ABB RobotStudio station: voice_control_abb.rspag

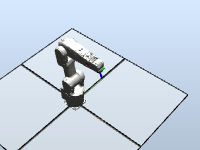
--- station ---
Station Station (saved by RobotStudio 6.7.7850.130)
Controller demo
  mechanical unit ROB_1: IRB1200_5_90_STD_02_2, 6 joints, base frame (0, 0, 0) mm
Layout (positions relative to the parent item):
  - IRB1200_5_90_STD_02_2 [mechanism, from Robots\IRB1200_5_90_STD_02.rslib] at (0, 0, 0) mm; joint values [-0.0263, -0.1564, 0.1446, 0.0099, 1.2195, -0.028] (rad or m)

--- Backups/demo/RAPID/TASK1/PROGMOD/Module1.mod ---
MODULE Module1
    PROC main()
        VAR socketdev server_socket;
        VAR socketdev client_socket;
        VAR string receiveStr;
        VAR string sReturn;
        VAR string recvStr{8};

        FOR i FROM 1 TO Dim(recvStr,1) DO
            recvStr{i}:=",";
        ENDFOR
        SocketCreate server_socket;
        SocketBind server_socket,"127.0.0.1",9000;
        SocketListen server_socket;
        SocketAccept server_socket,client_socket;
        SocketSend client_socket\Str:="Connected";
        TPErase;
        TPWrite "Connected";
        WHILE TRUE DO
            SocketReceive client_socket\Str:=receiveStr;
            TPWrite receiveStr;
            rSplitString receiveStr,recvStr;
            TEST recvStr{1}
            CASE "GetJ":
                cmd_GetJ recvStr,sReturn;
                SocketSend client_socket\Str:=sReturn;
            CASE "MoveJ":
                cmd_MoveJ recvStr,sReturn;
                SocketSend client_socket\Str:=sReturn;
            CASE "GetP":
                cmd_Getp recvStr,sReturn;
                SocketSend client_socket\Str:=sReturn;
            CASE "MoveL":
                cmd_MoveL recvStr,sReturn;
                SocketSend client_socket\Str:=sReturn;
            CASE "Forward":
                cmd_Forward recvStr,sReturn;
                SocketSend client_socket\Str:=sReturn;
            CASE "Backward":
                cmd_Backward recvStr,sReturn;
                SocketSend client_socket\Str:=sReturn;
            CASE "Left":
                cmd_Left recvStr,sReturn;
                SocketSend client_socket\Str:=sReturn;
            CASE "Right":
                cmd_Right recvStr,sReturn;
                SocketSend client_socket\Str:=sReturn;
            CASE "Up":
                cmd_Up recvStr,sReturn;
                SocketSend client_socket\Str:=sReturn;
            CASE "Down":
                cmd_Down recvStr,sReturn;
                SocketSend client_socket\Str:=sReturn;

            DEFAULT:
            ENDTEST
            WaitTime 0.1;
        ENDWHILE
        ERROR
            SocketClose server_socket;
            SocketClose client_socket;
            TPWrite "????";
        UNDO
    ENDPROC

    PROC cmd_GetJ(string recvStr{*},inout string sReturn)
        VAR jointtarget curJoint;
        curJoint:=CJointT();
        sReturn:=recvStr{1}+",0,";
        sReturn:=sReturn+NumToStr(curJoint.robax.rax_1,2)+",";
        sReturn:=sReturn+NumToStr(curJoint.robax.rax_2,2)+",";
        sReturn:=sReturn+NumToStr(curJoint.robax.rax_3,2)+",";
        sReturn:=sReturn+NumToStr(curJoint.robax.rax_4,2)+",";
        sReturn:=sReturn+NumToStr(curJoint.robax.rax_5,2)+",";
        sReturn:=sReturn+NumToStr(curJoint.robax.rax_6,2)+"/";
        ERROR
        sReturn:=recvStr{1}+",1/";
        TPWrite "error";
    ENDPROC

    PROC cmd_MoveJ(string recvStr{*},inout string sReturn)
        VAR jointtarget curJoint;
        VAR bool bResult;
        VAR num nJointValue{6};
        VAR num i;

        curJoint:=CJointT();
        bResult:=TRUE;
        FOR i FROM 1 TO Dim(recvStr,1)-2 DO
            bResult:=StrToVal(recvStr{i+1},nJointValue{i});
        ENDFOR

        curJoint.robax.rax_1:=nJointValue{1};
        curJoint.robax.rax_2:=nJointValue{2};
        curJoint.robax.rax_3:=nJointValue{3};
        curJoint.robax.rax_4:=nJointValue{4};
        curJoint.robax.rax_5:=nJointValue{5};
        curJoint.robax.rax_6:=nJointValue{6};
        MoveAbsJ curJoint,v1000,z50,tool0;
        sReturn:=recvStr{1}+",0/";
        ERROR
        sReturn:=recvStr{1}+",1/";
        TPWrite "error";

    ENDPROC

    PROC cmd_GetP(string recvStr{*},inout string sReturn)
        VAR robtarget curPoint;
        curPoint:=CRobT();
        sReturn:=recvStr{1}+",0,";
        sReturn:=sReturn+NumToStr(curPoint.trans.x,2)+",";
        sReturn:=sReturn+NumToStr(curPoint.trans.y,2)+",";
        sReturn:=sReturn+NumToStr(curPoint.trans.z,2)+",";
        sReturn:=sReturn+NumToStr(curPoint.rot.q1,2)+",";
        sReturn:=sReturn+NumToStr(curPoint.rot.q2,2)+",";
        sReturn:=sReturn+NumToStr(curPoint.rot.q3,2)+",";
        sReturn:=sReturn+NumToStr(curPoint.rot.q4,2)+"/";
        ERROR
        sReturn:=recvStr{1}+",1/";
        TPWrite "error";
    ENDPROC


    PROC cmd_MoveL(string recvStr{*},inout string sReturn)
        VAR robtarget curPoint;
        VAR bool bResult;
        VAR num nPointValue{7};
        VAR num i;

        curPoint:=CRobT();
        bResult:=TRUE;
        FOR i FROM 1 TO Dim(recvStr,1)-1 DO
            bResult:=StrToVal(recvStr{i+1},nPointValue{i});
        ENDFOR

        curPoint.trans.x:=nPointValue{1};
        curPoint.trans.y:=nPointValue{2};
        curPoint.trans.z:=nPointValue{3};
        curPoint.rot.q1:=nPointValue{4};
        curPoint.rot.q2:=nPointValue{5};
        curPoint.rot.q3:=nPointValue{6};
        curPoint.rot.q4:=nPointValue{7};
        MoveL curPoint,v1000,z50,tool0;
        sReturn:=recvStr{1}+",0/";
        ERROR
        sReturn:=recvStr{1}+",1/";
        TPWrite "error";

    ENDPROC


    PROC cmd_Forward(string recvStr{*},inout string sReturn)
        VAR robtarget curPoint;
        curPoint:=CRobT();
        curPoint:=Offs(curPoint,10,0,0);
        MoveL curPoint,v1000,z50,tool0;
        sReturn:=recvStr{1}+",0/";
        ERROR
        sReturn:=recvStr{1}+",1/";
        TPWrite "error";
    ENDPROC

    PROC cmd_Backward(string recvStr{*},inout string sReturn)
        VAR robtarget curPoint;
        curPoint:=CRobT();
        curPoint:=Offs(curPoint,-10,0,0);
        MoveL curPoint,v1000,z50,tool0;
        sReturn:=recvStr{1}+",0/";
        ERROR
        sReturn:=recvStr{1}+",1/";
        TPWrite "error";
    ENDPROC

    PROC cmd_Left(string recvStr{*},inout string sReturn)
        VAR robtarget curPoint;
        curPoint:=CRobT();
        curPoint:=Offs(curPoint,0,10,0);
        MoveL curPoint,v1000,z50,tool0;
        sReturn:=recvStr{1}+",0/";
        ERROR
        sReturn:=recvStr{1}+",1/";
        TPWrite "error";
    ENDPROC

    PROC cmd_Right(string recvStr{*},inout string sReturn)
        VAR robtarget curPoint;
        curPoint:=CRobT();
        curPoint:=Offs(curPoint,0,-10,0);
        MoveL curPoint,v1000,z50,tool0;
        sReturn:=recvStr{1}+",0/";
        ERROR
        sReturn:=recvStr{1}+",1/";
        TPWrite "error";
    ENDPROC

    PROC cmd_Up(string recvStr{*},inout string sReturn)
        VAR robtarget curPoint;
        curPoint:=CRobT();
        curPoint:=Offs(curPoint,0,0,10);
        MoveL curPoint,v1000,z50,tool0;
        sReturn:=recvStr{1}+",0/";
        ERROR
        sReturn:=recvStr{1}+",1/";
        TPWrite "error";
    ENDPROC

    PROC cmd_Down(string recvStr{*},inout string sReturn)
        VAR robtarget curPoint;
        curPoint:=CRobT();
        curPoint:=Offs(curPoint,0,0,-10);
        MoveL curPoint,v1000,z50,tool0;
        sReturn:=recvStr{1}+",0/";
        ERROR
        sReturn:=recvStr{1}+",1/";
        TPWrite "error";
    ENDPROC


    FUNC bool isCorrectStr(string strIn,inout string strOut)
        VAR num findNum;
        VAR bool bResult;

        findNum:=StrFind(strIn,1,"/");
        IF findNum>1 THEN
            bResult:=TRUE;
            strOut:=StrPart(strIn,1,findNum-1);
        ELSE
            bResult:=False;
        ENDIF

        RETURN bResult;
    ENDFUNC

  PROC rSplitString(string strIn,INOUT string strOut{*})
    VAR num str_Len;
        VAR num startBit;
        VAR num endBit;
        VAR num i;
        VAR string newStr;
        VAR bool bResult;

        startBit:=1;
        endBit:=1;
        i:=1;

        bResult:=isCorrectStr(strIn,newStr);
        IF bResult THEN
            WHILE StrFind(newStr,startBit,",")<>StrLen(newStr)+1 DO
                str_Len:=StrLen(newStr);
                endBit:=StrFind(newStr,startBit,",");
                strOut{i}:=StrPart(newStr,startBit,endBit-1);

                newStr:=StrPart(newStr,endBit+1,str_Len-endBit);
                i:=i+1;
            ENDWHILE
            bResult:=isCorrectStr(newStr,newStr);
            strOut{i}:=newStr;
        ENDIF
  ENDPROC

ENDMODULE
